// TIA Portal V21 export
FUNCTION_BLOCK "MotorSim"   // FB4, LAD
{ S7_Optimized_Access := 'TRUE' }
// stored: MemoryReserve 100, SetENOAutomatically false
   VAR_INPUT
      fwd : Bool;
      rev : Bool;
      simFault : Bool;
      speedSp : Real;
   END_VAR
   VAR_OUTPUT
      fbFwd : Bool;
      fbRev : Bool;
      speedPv : Real;
      fault : Bool;
   END_VAR
   VAR
      fwdTimer : TON_TIME;
      revTimer : TON_TIME;
      lag { S7_SetPoint := 'True'} : Filter_PT1;
   END_VAR
   // lag.Lag := 4.0;
BEGIN

REGION Network 1
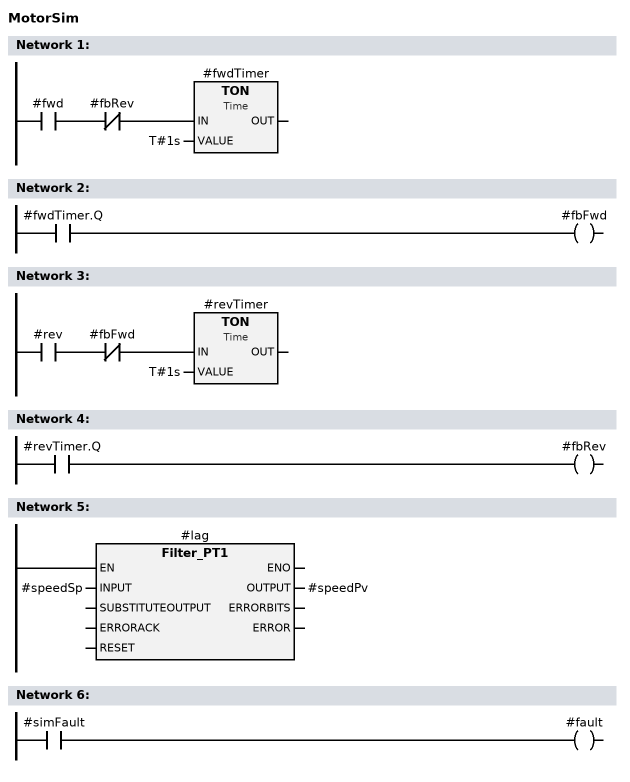
   #fwdTimer(IN := #fwd AND NOT #fbRev, PT := T#1s);   // TON coil
END_REGION

REGION Network 2
   RUNG wire#powerrail
      Contact( #fwdTimer.Q )
      Coil( #fbFwd )
   END_RUNG
   // the same network as SCL:
   #fbFwd := #fwdTimer.Q;
END_REGION

REGION Network 3
   #revTimer(IN := #rev AND NOT #fbFwd, PT := T#1s);   // TON coil
END_REGION

REGION Network 4
   RUNG wire#powerrail
      Contact( #revTimer.Q )
      Coil( #fbRev )
   END_RUNG
   // the same network as SCL:
   #fbRev := #revTimer.Q;
END_REGION

REGION Network 5
   RUNG wire#powerrail
      #lag.Filter_PT1(Input := #speedSp, SubstituteOutput :=, ErrorAck :=, Reset :=, Output => #speedPv, ErrorBits =>, Error =>)
   END_RUNG
   // the same network as SCL:
   #lag(Input := #speedSp, Output => #speedPv);   // Filter_PT1
END_REGION

REGION Network 6
   RUNG wire#powerrail
      Contact( #simFault )
      Coil( #fault )
   END_RUNG
   // the same network as SCL:
   #fault := #simFault;
END_REGION
END_FUNCTION_BLOCK
